Fanuc TP program (LS listing): PICKFRAME.LS

/PROG  PICKFRAME
/ATTR
OWNER		= MNEDITOR;
COMMENT		= "macro Frame chae";
PROG_SIZE	= 187;
CREATE		= DATE 19-12-17  TIME 17:35:26;
MODIFIED	= DATE 19-12-17  TIME 17:36:00;
FILE_NAME	= ;
VERSION		= 0;
LINE_COUNT	= 2;
MEMORY_SIZE	= 551;
PROTECT		= READ_WRITE;
TCD:  STACK_SIZE	= 0,
      TASK_PRIORITY	= 50,
      TIME_SLICE	= 0,
      BUSY_LAMP_OFF	= 0,
      ABORT_REQUEST	= 0,
      PAUSE_REQUEST	= 0;
DEFAULT_GROUP	= 1,*,*,*,*;
CONTROL_CODE	= 00000000 00000000;
/APPL
/APPL

AUTO_SINGULARITY_HEADER;
  ENABLE_SINGULARITY_AVOIDANCE   : TRUE;
/MN
   1:  UFRAME_NUM=1 ;
   2:  UTOOL_NUM=1 ;
/POS
/END
